(* PLC project PLC_ODOT.project, CODESYS CODESYS V3.5 SP19 *)
(* stored: creationDateTime 2026-01-26T16:58:28.1301043, modificationDateTime 2026-01-26T16:51:59.9229809 *)

FUNCTION_BLOCK FbScale
  VAR_INPUT
    In : REAL := 0;  (* Вход до масштабирования. *)
    InMax : REAL := 27648;  (* Максимум входного диапазона. *)
    InMin : REAL := 0;  (* Минимум входного диапазона. *)
    OutMax : REAL := 20;  (* Максимум выходного диапазона. *)
    OutMin : REAL := 4;  (* Минимум выходного диапазона. *)
  END_VAR
  VAR_OUTPUT
    Out : REAL := 0;  (* Выход после масштабирования. *)
  END_VAR

            //       DbScale
//    +-----------+
//    |  FbScale  |
// ->-|In      Out|->-
//   -|InMax      |
//   -|InMin      |
//   -|OutMax     |
//   -|OutMin     |
//    +-----------+

//Масштабирование сигнала.
IF (InMax = InMin) THEN //Деление на 0 может остановить процессор.
//При ошибке исходных данных.
Out := 0.0;
ELSE
//Масштабирование.
Out := (OutMax - OutMin) * ((In - InMin)/(InMax - InMin)) + OutMin;
END_IF;


// Статическая характеристика.
//
//       ^ Out
//       |
// OutMax|<---------------*
//       |              * |
//       |            *   |
//    Out|<---------*     |
//       |        * |     |
//       |      *   |     |
// OutMin|<---*     |     |
//       |    |     |     |
//       |    |     |     |
//       +---------------------> In
//          InMin  In   InMax

// Выход сигнал
// Out = k * In + b
//
// Для расчета k, b надо решить систему двух линейных уравнений с двумя неизвестными.
// {OutMax = k * InMax + b
// {OutMin = k * InMin + b
//
// Усиление:
//      OutMax - OutMin 
// k = -----------------
//       InMax - InMin  
//
// Смещение:
// b = OutMax - k * InMax
//
// После подстановки в уравнение Out = k * In + b констант k, b,
// и сокращения числа арифметических операций до минимума получаем:
// Out := (OutMax - OutMin) * ((In - InMin)/(InMax - InMin)) + OutMin;

// Данное линейное преобразование на практике легко вывести через промежуточный диаппазон 0...1:
// InMin...InMax -> 0...(InMax-InMin) -> 0...1 -> 0...(OutMax-OutMin) -> OutMin...OutMax.
// Пример рассчета давления с датчика  4...20мА -> 0...10Бар.
// 4...20 -  4 = 0...16
// 0...16 / 16 = 0...1
// 0...1  * 10 = 0...10
// При токе 12мА
// 12  -   4 = 8
// 8   /  16 = 0.5
// 0.5 *  10 = 5Бар
// Давление 5Бар.

//  +---------+
//  | GNU GPL |
//  +---------+
//  |
//  |
//  .= .-_-. =.
// ((_/)o o(\_))
//  `-'(. .)`-'
//  |/| \_/ |\
//  ( |     | )
//  /"\_____/"\
//  \__)   (__/
// @COPYLEFT ALL WRONGS RESERVED :)
// Author: VA
// Contacts: DIY.PLC.314@gmail.com
// License: GNU GPL v2
//
// https://www.youtube.com/@DIY_PLC
// https://github.com/DIYPLC

          
END_FUNCTION_BLOCK
